Fanuc KAREL source: kt00888.KL

-- PROVISIONAL review KL for V940-1; original PC SHA256 5ceda6acda4be157b80006e7a857ab8388dcf0d98c2570018be5126b5e01196a
-- Incomplete behavior may be omitted. Consult companion uncertainty JSON. Do not deploy.
PROGRAM KT00888
%NOLOCKGROUP
-- UNRESOLVED_DECL P1 type=000101
-- UNRESOLVED_DECL P2 type=000101
-- UNRESOLVED_DECL OUT type=000101
BEGIN
  -- V9_ZERO_TABLE_METADATA_HINT layout=0001; no indexed target words; source/name/runtime held
  -- UNRESOLVED_PC offsets 5-32; opcodes 27,22,1C,76,7E,4A
  -- UNRESOLVED_PC offsets 37-41; opcodes 7F
END KT00888
